// TIA Portal V15.1 export
// export: Created 2020-06-12T07:35:48.4287109Z, ExportSetting None, DisplayName Totally Integrated Automation Portal, DisplayVersion V15.1, DisplayName TIA Portal Openness, DisplayVersion V15.1, DisplayName STEP 7 Professional, DisplayVersion V15.1, DisplayName STEP 7 Safety, DisplayVersion V15.1, DisplayName WinCC Advanced, DisplayVersion V15.1
FUNCTION "PWR_call" : Void   // FC79, FBD
TITLE = Melt Power supply
{ S7_Optimized_Access := 'TRUE' }
// stored: SetENOAutomatically False
BEGIN

REGION Network 1: Trafo control
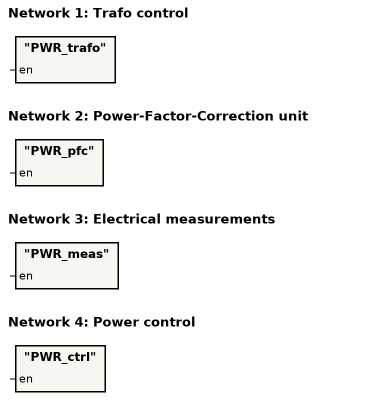
   "PWR_trafo"();
END_REGION

REGION Network 2: Power-Factor-Correction unit
   "PWR_pfc"();
END_REGION

REGION Network 3: Electrical measurements
   "PWR_meas"();
END_REGION

REGION Network 4: Power control
   "PWR_ctrl"();
END_REGION
END_FUNCTION
